INTERFACE ITF_EM_Infeed_Checkweigher

END_INTERFACE

(* stored: Version 1.1.0.1, ProductVersion 3.1.4024.12
   Itf ITF_EM_Infeed_Checkweigher: Id {ea284206-aee2-406e-9690-49de684e8e91} *)
